(* PLC project Scenario7v1_Final.project, CODESYS CODESYS V3.5 SP5 Patch 1 *)
(* stored: creationDateTime 2014-09-12T06:04:18.7394832, modificationDateTime 2014-09-11T21:24:11.718058 *)

FUNCTION_BLOCK Magazin
  VAR_INPUT
    SliderNotMovedOut : BOOL;
    SliderMovedOut : BOOL;
    WorkpieceReady : BOOL;
    CraneDown : BOOL;
    CraneUp : BOOL;
    CraneOnConveyor : BOOL;
    CraneOnMagazin : BOOL;
    CraneSucked : BOOL;
    StartButtonMagazin : BOOL;
    SFCReset : BOOL;
    StartVar : BOOL;
  END_VAR
  VAR_OUTPUT
    CraneLower : BOOL;
    MagazinVacuumOff : BOOL;
    MagazinVacuumOn : BOOL;
    CraneTurnCounterclockwise : BOOL;
    CraneTurnClockwise : BOOL;
    MagazinSlider : BOOL;
    MagazinGreenLamp : BOOL;
    MagazinWhiteLamp : BOOL;
    StartCommandMagazin : BOOL;
  END_VAR
  VAR
    interconnectMagazinStartCommand : BOOL;
    SFCInit : BOOL;
  END_VAR

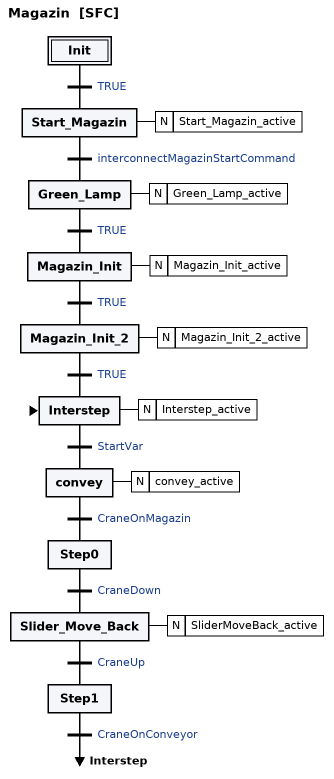
INITIAL_STEP Init:
END_STEP
TRANSITION FROM Init TO Start_Magazin
  := TRUE;
END_TRANSITION
STEP Start_Magazin:
  Start_Magazin_active(N);
END_STEP
TRANSITION FROM Start_Magazin TO Green_Lamp
  := interconnectMagazinStartCommand;
END_TRANSITION
STEP Green_Lamp:
  Green_Lamp_active(N);
END_STEP
TRANSITION FROM Green_Lamp TO Magazin_Init
  := TRUE;
END_TRANSITION
STEP Magazin_Init:
  Magazin_Init_active(N);
END_STEP
TRANSITION FROM Magazin_Init TO Magazin_Init_2
  := TRUE;
END_TRANSITION
STEP Magazin_Init_2:
  Magazin_Init_2_active(N);
END_STEP
TRANSITION FROM Magazin_Init_2 TO Interstep
  := TRUE;
END_TRANSITION
STEP Interstep:
  Interstep_active(N);
END_STEP
TRANSITION FROM Interstep TO convey
  := StartVar;
END_TRANSITION
STEP convey:
  convey_active(N);
END_STEP
TRANSITION FROM convey TO Step0
  := CraneOnMagazin;
END_TRANSITION
STEP Step0:
END_STEP
TRANSITION FROM Step0 TO Slider_Move_Back
  := CraneDown;
END_TRANSITION
STEP Slider_Move_Back:
  SliderMoveBack_active(N);
END_STEP
TRANSITION FROM Slider_Move_Back TO Step1
  := CraneUp;
END_TRANSITION
STEP Step1:
END_STEP
TRANSITION FROM Step1 TO Interstep
  := CraneOnConveyor;
END_TRANSITION

ACTION Magazin_Init_active:
                MagazinSlider := TRUE;
              
END_ACTION

ACTION Start_Magazin_active:
                MagazinSlider := FALSE;
MagazinGreenLamp := FALSE;
StartVar := FALSE;
StartCommandMagazin := FALSE;


IF(StartButtonMagazin = TRUE) THEN
	interconnectMagazinStartCommand := TRUE;
END_IF
              
END_ACTION

ACTION Green_Lamp_active:
                MagazinGreenLamp := TRUE;
interconnectMagazinStartCommand := FALSE;
              
END_ACTION

ACTION convey_active:
                IF(SliderNotMovedOut)THEN
	MagazinSlider := TRUE;
END_IF
              
END_ACTION

ACTION SliderMoveBack_active:
                IF((SliderMovedOut = TRUE)AND(SliderNotMovedOut = FALSE))THEN
	MagazinSlider := FALSE;
END_IF
              
END_ACTION

ACTION Magazin_Init_2_active:
                MagazinSlider := FALSE;
              
END_ACTION

ACTION Interstep_active:
                StartCommandMagazin := TRUE;
              
END_ACTION
END_FUNCTION_BLOCK

FUNCTION_BLOCK Stamp
  VAR_INPUT
    StampSliderSensorMovedOut : BOOL;
    StampSliderSensorMovedIn : BOOL;
    StampSliderFilled : BOOL;
    StampUp : BOOL;
    StampLowered : BOOL;
    CraneDown : BOOL;
    CraneUp : BOOL;
    CraneSucked : BOOL;
    CranePositionStamp : BOOL;
    CraneOnConveyor : BOOL;
    StampStartButton : BOOL;
    SFCReset : BOOL;
    StartVar : BOOL;
  END_VAR
  VAR_OUTPUT
    StampSliderMovedOut : BOOL;
    StampSliderMovedIn : BOOL;
    StampWhiteLamp : BOOL;
    StampPusher : BOOL;
    StampGreenLamp : BOOL;
    StampPressure : BOOL;
    StartCommandStamp : BOOL;
  END_VAR
  VAR
    interconnect : BOOL;
    Timer : TON;
    Duration : TIME := TIME#500ms;
    interconnectStampStartCommand : BOOL;
    SFCInit : BOOL;
  END_VAR

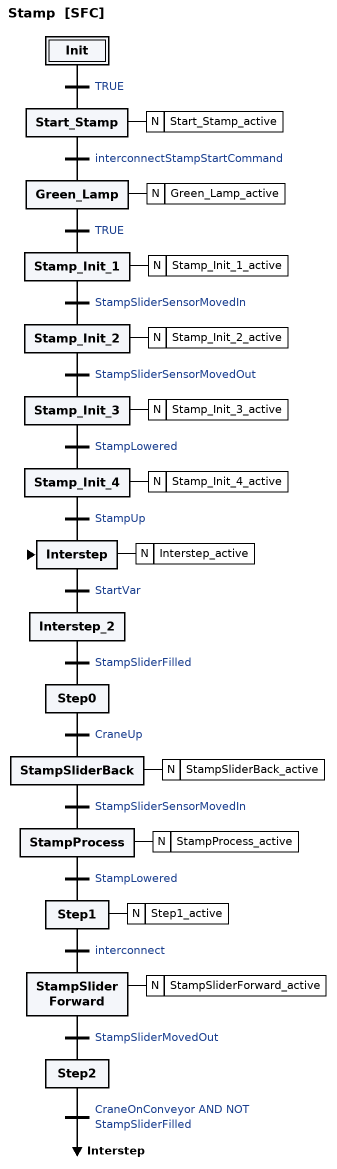
INITIAL_STEP Init:
END_STEP
TRANSITION FROM Init TO Start_Stamp
  := TRUE;
END_TRANSITION
STEP Start_Stamp:
  Start_Stamp_active(N);
END_STEP
TRANSITION FROM Start_Stamp TO Green_Lamp
  := interconnectStampStartCommand;
END_TRANSITION
STEP Green_Lamp:
  Green_Lamp_active(N);
END_STEP
TRANSITION FROM Green_Lamp TO Stamp_Init_1
  := TRUE;
END_TRANSITION
STEP Stamp_Init_1:
  Stamp_Init_1_active(N);
END_STEP
TRANSITION FROM Stamp_Init_1 TO Stamp_Init_2
  := StampSliderSensorMovedIn;
END_TRANSITION
STEP Stamp_Init_2:
  Stamp_Init_2_active(N);
END_STEP
TRANSITION FROM Stamp_Init_2 TO Stamp_Init_3
  := StampSliderSensorMovedOut;
END_TRANSITION
STEP Stamp_Init_3:
  Stamp_Init_3_active(N);
END_STEP
TRANSITION FROM Stamp_Init_3 TO Stamp_Init_4
  := StampLowered;
END_TRANSITION
STEP Stamp_Init_4:
  Stamp_Init_4_active(N);
END_STEP
TRANSITION FROM Stamp_Init_4 TO Interstep
  := StampUp;
END_TRANSITION
STEP Interstep:
  Interstep_active(N);
END_STEP
TRANSITION FROM Interstep TO Interstep_2
  := StartVar;
END_TRANSITION
STEP Interstep_2:
END_STEP
TRANSITION FROM Interstep_2 TO Step0
  := StampSliderFilled;
END_TRANSITION
STEP Step0:
END_STEP
TRANSITION FROM Step0 TO StampSliderBack
  := CraneUp;
END_TRANSITION
STEP StampSliderBack:
  StampSliderBack_active(N);
END_STEP
TRANSITION FROM StampSliderBack TO StampProcess
  := StampSliderSensorMovedIn;
END_TRANSITION
STEP StampProcess:
  StampProcess_active(N);
END_STEP
TRANSITION FROM StampProcess TO Step1
  := StampLowered;
END_TRANSITION
STEP Step1:
  Step1_active(N);
END_STEP
TRANSITION FROM Step1 TO StampSliderForward
  := interconnect;
END_TRANSITION
STEP StampSliderForward:
  StampSliderForward_active(N);
END_STEP
TRANSITION FROM StampSliderForward TO Step2
  := StampSliderMovedOut;
END_TRANSITION
STEP Step2:
END_STEP
TRANSITION FROM Step2 TO Interstep
  := CraneOnConveyor AND NOT StampSliderFilled;
END_TRANSITION

ACTION Start_Stamp_active:
                StampSliderMovedOut := FALSE;
StampSliderMovedIn := FALSE;
StampPusher := FALSE;
StampGreenLamp := FALSE;
StampPressure := FALSE;
StartCommandStamp := FALSE;


IF(StampStartButton = TRUE) THEN
	interconnectStampStartCommand := TRUE;
END_IF
              
END_ACTION

ACTION StampSliderForward_active:
                StampPusher := FALSE;
StampSliderMovedOut := TRUE;

IF((StampLowered=FALSE)AND(StampUp=TRUE))THEN
	interconnect := FALSE;
END_IF

Timer(IN:=FALSE, PT:=T#1ms);
              
END_ACTION

ACTION StampSliderBack_active:
                StampSliderMovedIn := TRUE;
StampSliderMovedOut := FALSE;
              
END_ACTION

ACTION Stamp_Init_1_active:
                StampSliderMovedIn := TRUE;
StampSliderMovedOut := FALSE;
              
END_ACTION

ACTION Step1_active:
                Timer(IN:=StampLowered, PT:=T#500MS);
interconnect := Timer.Q;
              
END_ACTION

ACTION Interstep_active:
                StartCommandStamp := TRUE;
              
END_ACTION

ACTION Green_Lamp_active:
                StampGreenLamp := TRUE;
interconnectStampStartCommand := FALSE;
              
END_ACTION

ACTION Stamp_Init_4_active:
                StampPusher := FALSE;
              
END_ACTION

ACTION Stamp_Init_3_active:
                StampPusher := TRUE;
              
END_ACTION

ACTION Stamp_Init_2_active:
                StampSliderMovedIn := FALSE;
StampSliderMovedOut := TRUE;
              
END_ACTION

ACTION StampProcess_active:
                StampSliderMovedIn := FALSE;
StampPusher := TRUE;
              
END_ACTION
END_FUNCTION_BLOCK

FUNCTION_BLOCK Crane
  VAR_INPUT
    SliderNotMovedOut : BOOL;
    SliderMovedOut : BOOL;
    MagazinCapacitiveSensor : BOOL;
    WorkpieceReady : BOOL;
    CraneDown : BOOL;
    CraneUp : BOOL;
    CraneOnConveyor : BOOL;
    CraneOnMagazin : BOOL;
    CraneSucked : BOOL;
    StampLowered : BOOL;
    CranePositionStamp : BOOL;
    MagazinOpticalSensor : BOOL;
    StampSliderFilled : BOOL;
    StartButtonMagazin : BOOL;
    SFCReset : BOOL;
    StartVar : BOOL;
    StampSliderSensorMovedOut : BOOL;
  END_VAR
  VAR_OUTPUT
    CraneLower : BOOL;
    MagazinVacuumOff : BOOL;
    MagazinVacuumOn : BOOL;
    CraneTurnCounterclockwise : BOOL;
    CraneTurnClockwise : BOOL;
    StartCommandCrane : BOOL;
  END_VAR
  VAR
    Timer1 : TON;
    Duration1 : TIME := TIME#1s500ms;
    actualtime1 : TIME;
    interconnect : BOOL;
    interconnectCraneStartCommand : BOOL;
    TimeDelay_Timer : TON;
    TimeDelay_Timer_Duration : TIME := TIME#50ms;
    TimeDelay_Timer_interconnect : BOOL;
    SFCInit : BOOL;
  END_VAR

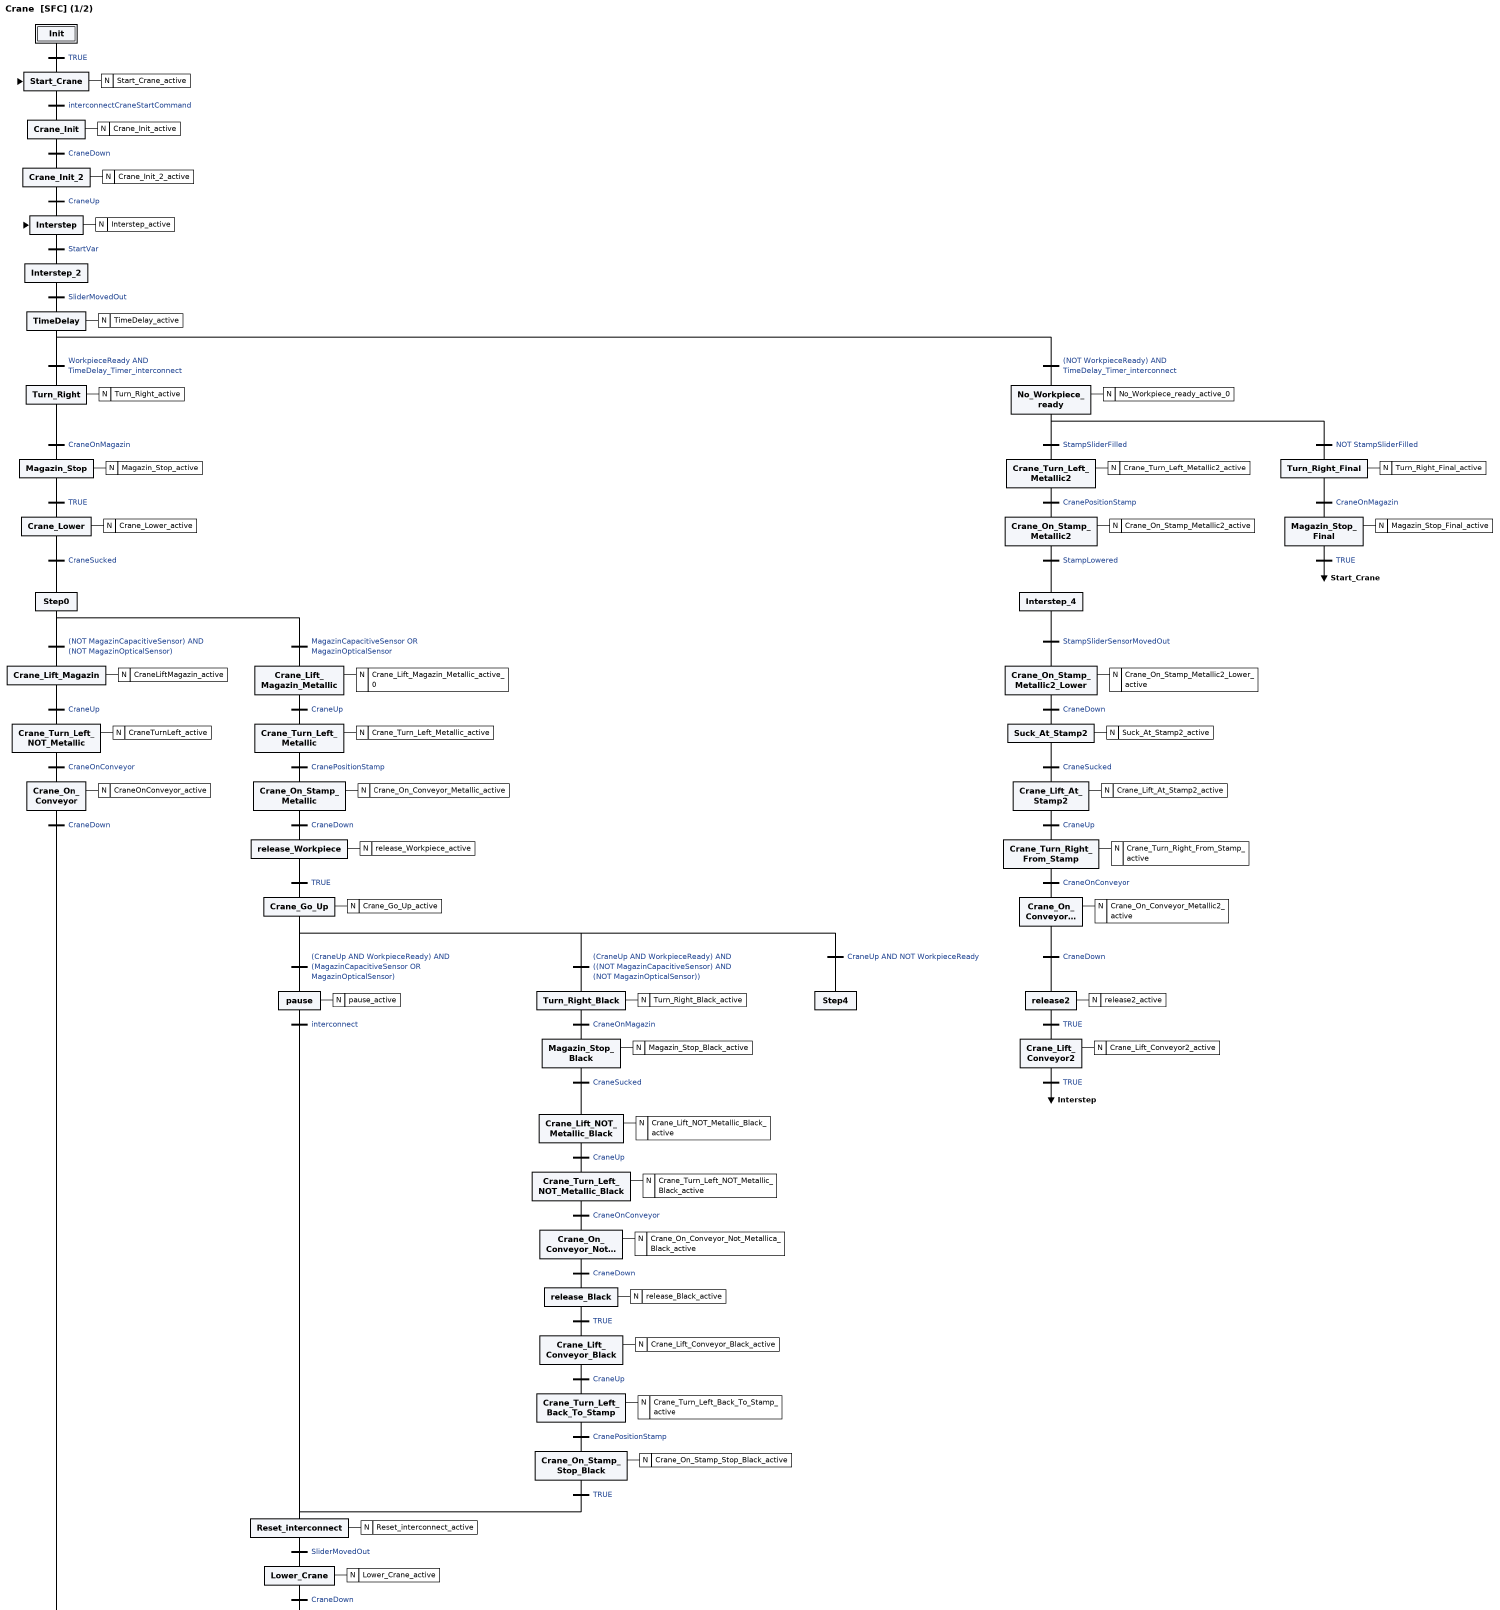
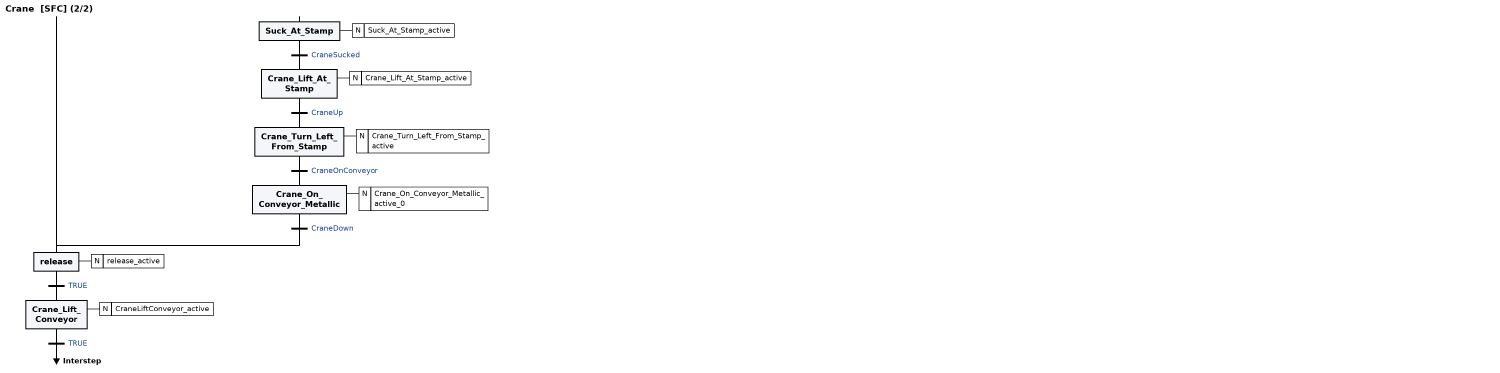
INITIAL_STEP Init:
END_STEP
TRANSITION FROM Init TO Start_Crane
  := TRUE;
END_TRANSITION
STEP Start_Crane:
  Start_Crane_active(N);
END_STEP
TRANSITION FROM Start_Crane TO Crane_Init
  := interconnectCraneStartCommand;
END_TRANSITION
STEP Crane_Init:
  Crane_Init_active(N);
END_STEP
TRANSITION FROM Crane_Init TO Crane_Init_2
  := CraneDown;
END_TRANSITION
STEP Crane_Init_2:
  Crane_Init_2_active(N);
END_STEP
TRANSITION FROM Crane_Init_2 TO Interstep
  := CraneUp;
END_TRANSITION
STEP Interstep:
  Interstep_active(N);
END_STEP
TRANSITION FROM Interstep TO Interstep_2
  := StartVar;
END_TRANSITION
STEP Interstep_2:
END_STEP
TRANSITION FROM Interstep_2 TO TimeDelay
  := SliderMovedOut;
END_TRANSITION
STEP TimeDelay:
  TimeDelay_active(N);
END_STEP
TRANSITION FROM TimeDelay TO Turn_Right
  := WorkpieceReady AND TimeDelay_Timer_interconnect;
END_TRANSITION
TRANSITION FROM TimeDelay TO No_Workpiece_ready
  := (NOT WorkpieceReady) AND TimeDelay_Timer_interconnect;
END_TRANSITION
STEP Turn_Right:
  Turn_Right_active(N);
END_STEP
TRANSITION FROM Turn_Right TO Magazin_Stop
  := CraneOnMagazin;
END_TRANSITION
STEP Magazin_Stop:
  Magazin_Stop_active(N);
END_STEP
TRANSITION FROM Magazin_Stop TO Crane_Lower
  := TRUE;
END_TRANSITION
STEP Crane_Lower:
  Crane_Lower_active(N);
END_STEP
TRANSITION FROM Crane_Lower TO Step0
  := CraneSucked;
END_TRANSITION
STEP Step0:
END_STEP
TRANSITION FROM Step0 TO Crane_Lift_Magazin
  := (NOT MagazinCapacitiveSensor) AND (NOT MagazinOpticalSensor);
END_TRANSITION
TRANSITION FROM Step0 TO Crane_Lift_Magazin_Metallic
  := MagazinCapacitiveSensor OR MagazinOpticalSensor;
END_TRANSITION
STEP Crane_Lift_Magazin:
  CraneLiftMagazin_active(N);
END_STEP
TRANSITION FROM Crane_Lift_Magazin TO Crane_Turn_Left_NOT_Metallic
  := CraneUp;
END_TRANSITION
STEP Crane_Turn_Left_NOT_Metallic:
  CraneTurnLeft_active(N);
END_STEP
TRANSITION FROM Crane_Turn_Left_NOT_Metallic TO Crane_On_Conveyor
  := CraneOnConveyor;
END_TRANSITION
STEP Crane_On_Conveyor:
  CraneOnConveyor_active(N);
END_STEP
TRANSITION FROM Crane_On_Conveyor TO release
  := CraneDown;
END_TRANSITION
STEP Crane_Lift_Magazin_Metallic:
  Crane_Lift_Magazin_Metallic_active_0(N);
END_STEP
TRANSITION FROM Crane_Lift_Magazin_Metallic TO Crane_Turn_Left_Metallic
  := CraneUp;
END_TRANSITION
STEP Crane_Turn_Left_Metallic:
  Crane_Turn_Left_Metallic_active(N);
END_STEP
TRANSITION FROM Crane_Turn_Left_Metallic TO Crane_On_Stamp_Metallic
  := CranePositionStamp;
END_TRANSITION
STEP Crane_On_Stamp_Metallic:
  Crane_On_Conveyor_Metallic_active(N);
END_STEP
TRANSITION FROM Crane_On_Stamp_Metallic TO release_Workpiece
  := CraneDown;
END_TRANSITION
STEP release_Workpiece:
  release_Workpiece_active(N);
END_STEP
TRANSITION FROM release_Workpiece TO Crane_Go_Up
  := TRUE;
END_TRANSITION
STEP Crane_Go_Up:
  Crane_Go_Up_active(N);
END_STEP
TRANSITION FROM Crane_Go_Up TO pause
  := (CraneUp AND WorkpieceReady) AND (MagazinCapacitiveSensor OR MagazinOpticalSensor);
END_TRANSITION
TRANSITION FROM Crane_Go_Up TO Turn_Right_Black
  := (CraneUp AND WorkpieceReady) AND ((NOT MagazinCapacitiveSensor) AND (NOT MagazinOpticalSensor));
END_TRANSITION
TRANSITION FROM Crane_Go_Up TO Step4
  := CraneUp AND NOT WorkpieceReady;
END_TRANSITION
STEP pause:
  pause_active(N);
END_STEP
TRANSITION FROM pause TO Reset_interconnect
  := interconnect;
END_TRANSITION
STEP Turn_Right_Black:
  Turn_Right_Black_active(N);
END_STEP
TRANSITION FROM Turn_Right_Black TO Magazin_Stop_Black
  := CraneOnMagazin;
END_TRANSITION
STEP Magazin_Stop_Black:
  Magazin_Stop_Black_active(N);
END_STEP
TRANSITION FROM Magazin_Stop_Black TO Crane_Lift_NOT_Metallic_Black
  := CraneSucked;
END_TRANSITION
STEP Crane_Lift_NOT_Metallic_Black:
  Crane_Lift_NOT_Metallic_Black_active(N);
END_STEP
TRANSITION FROM Crane_Lift_NOT_Metallic_Black TO Crane_Turn_Left_NOT_Metallic_Black
  := CraneUp;
END_TRANSITION
STEP Crane_Turn_Left_NOT_Metallic_Black:
  Crane_Turn_Left_NOT_Metallic_Black_active(N);
END_STEP
TRANSITION FROM Crane_Turn_Left_NOT_Metallic_Black TO Crane_On_Conveyor_Not_Metallica_Black
  := CraneOnConveyor;
END_TRANSITION
STEP Crane_On_Conveyor_Not_Metallica_Black:
  Crane_On_Conveyor_Not_Metallica_Black_active(N);
END_STEP
TRANSITION FROM Crane_On_Conveyor_Not_Metallica_Black TO release_Black
  := CraneDown;
END_TRANSITION
STEP release_Black:
  release_Black_active(N);
END_STEP
TRANSITION FROM release_Black TO Crane_Lift_Conveyor_Black
  := TRUE;
END_TRANSITION
STEP Crane_Lift_Conveyor_Black:
  Crane_Lift_Conveyor_Black_active(N);
END_STEP
TRANSITION FROM Crane_Lift_Conveyor_Black TO Crane_Turn_Left_Back_To_Stamp
  := CraneUp;
END_TRANSITION
STEP Crane_Turn_Left_Back_To_Stamp:
  Crane_Turn_Left_Back_To_Stamp_active(N);
END_STEP
TRANSITION FROM Crane_Turn_Left_Back_To_Stamp TO Crane_On_Stamp_Stop_Black
  := CranePositionStamp;
END_TRANSITION
STEP Crane_On_Stamp_Stop_Black:
  Crane_On_Stamp_Stop_Black_active(N);
END_STEP
TRANSITION FROM Crane_On_Stamp_Stop_Black TO Reset_interconnect
  := TRUE;
END_TRANSITION
STEP Step4:
END_STEP
STEP Reset_interconnect:
  Reset_interconnect_active(N);
END_STEP
TRANSITION FROM Reset_interconnect TO Lower_Crane
  := SliderMovedOut;
END_TRANSITION
STEP Lower_Crane:
  Lower_Crane_active(N);
END_STEP
TRANSITION FROM Lower_Crane TO Suck_At_Stamp
  := CraneDown;
END_TRANSITION
STEP Suck_At_Stamp:
  Suck_At_Stamp_active(N);
END_STEP
TRANSITION FROM Suck_At_Stamp TO Crane_Lift_At_Stamp
  := CraneSucked;
END_TRANSITION
STEP Crane_Lift_At_Stamp:
  Crane_Lift_At_Stamp_active(N);
END_STEP
TRANSITION FROM Crane_Lift_At_Stamp TO Crane_Turn_Left_From_Stamp
  := CraneUp;
END_TRANSITION
STEP Crane_Turn_Left_From_Stamp:
  Crane_Turn_Left_From_Stamp_active(N);
END_STEP
TRANSITION FROM Crane_Turn_Left_From_Stamp TO Crane_On_Conveyor_Metallic
  := CraneOnConveyor;
END_TRANSITION
STEP Crane_On_Conveyor_Metallic:
  Crane_On_Conveyor_Metallic_active_0(N);
END_STEP
TRANSITION FROM Crane_On_Conveyor_Metallic TO release
  := CraneDown;
END_TRANSITION
STEP release:
  release_active(N);
END_STEP
TRANSITION FROM release TO Crane_Lift_Conveyor
  := TRUE;
END_TRANSITION
STEP Crane_Lift_Conveyor:
  CraneLiftConveyor_active(N);
END_STEP
TRANSITION FROM Crane_Lift_Conveyor TO Interstep
  := TRUE;
END_TRANSITION
STEP No_Workpiece_ready:
  No_Workpiece_ready_active_0(N);
END_STEP
TRANSITION FROM No_Workpiece_ready TO Crane_Turn_Left_Metallic2
  := StampSliderFilled;
END_TRANSITION
TRANSITION FROM No_Workpiece_ready TO Turn_Right_Final
  := NOT StampSliderFilled;
END_TRANSITION
STEP Crane_Turn_Left_Metallic2:
  Crane_Turn_Left_Metallic2_active(N);
END_STEP
TRANSITION FROM Crane_Turn_Left_Metallic2 TO Crane_On_Stamp_Metallic2
  := CranePositionStamp;
END_TRANSITION
STEP Crane_On_Stamp_Metallic2:
  Crane_On_Stamp_Metallic2_active(N);
END_STEP
TRANSITION FROM Crane_On_Stamp_Metallic2 TO Interstep_4
  := StampLowered;
END_TRANSITION
STEP Interstep_4:
END_STEP
TRANSITION FROM Interstep_4 TO Crane_On_Stamp_Metallic2_Lower
  := StampSliderSensorMovedOut;
END_TRANSITION
STEP Crane_On_Stamp_Metallic2_Lower:
  Crane_On_Stamp_Metallic2_Lower_active(N);
END_STEP
TRANSITION FROM Crane_On_Stamp_Metallic2_Lower TO Suck_At_Stamp2
  := CraneDown;
END_TRANSITION
STEP Suck_At_Stamp2:
  Suck_At_Stamp2_active(N);
END_STEP
TRANSITION FROM Suck_At_Stamp2 TO Crane_Lift_At_Stamp2
  := CraneSucked;
END_TRANSITION
STEP Crane_Lift_At_Stamp2:
  Crane_Lift_At_Stamp2_active(N);
END_STEP
TRANSITION FROM Crane_Lift_At_Stamp2 TO Crane_Turn_Right_From_Stamp
  := CraneUp;
END_TRANSITION
STEP Crane_Turn_Right_From_Stamp:
  Crane_Turn_Right_From_Stamp_active(N);
END_STEP
TRANSITION FROM Crane_Turn_Right_From_Stamp TO Crane_On_Conveyor_Metallic2
  := CraneOnConveyor;
END_TRANSITION
STEP Crane_On_Conveyor_Metallic2:
  Crane_On_Conveyor_Metallic2_active(N);
END_STEP
TRANSITION FROM Crane_On_Conveyor_Metallic2 TO release2
  := CraneDown;
END_TRANSITION
STEP release2:
  release2_active(N);
END_STEP
TRANSITION FROM release2 TO Crane_Lift_Conveyor2
  := TRUE;
END_TRANSITION
STEP Crane_Lift_Conveyor2:
  Crane_Lift_Conveyor2_active(N);
END_STEP
TRANSITION FROM Crane_Lift_Conveyor2 TO Interstep
  := TRUE;
END_TRANSITION
STEP Turn_Right_Final:
  Turn_Right_Final_active(N);
END_STEP
TRANSITION FROM Turn_Right_Final TO Magazin_Stop_Final
  := CraneOnMagazin;
END_TRANSITION
STEP Magazin_Stop_Final:
  Magazin_Stop_Final_active(N);
END_STEP
TRANSITION FROM Magazin_Stop_Final TO Start_Crane
  := TRUE;
END_TRANSITION

ACTION Interstep_active:
                StartCommandCrane := TRUE;
              
END_ACTION

ACTION Crane_Lift_NOT_Metallic_Black_active:
                CraneLower := FALSE;
              
END_ACTION

ACTION Suck_At_Stamp_active:
                MagazinVacuumOn := TRUE;
MagazinVacuumOff := FALSE;
              
END_ACTION

ACTION Magazin_Stop_Black_active:
                CraneTurnClockwise := FALSE;
CraneTurnCounterclockwise := FALSE;
MagazinVacuumOn := TRUE;
MagazinVacuumOff := FALSE;
CraneLower := TRUE;
              
END_ACTION

ACTION Crane_On_Conveyor_Not_Metallica_Black_active:
                CraneTurnCounterclockwise := FALSE;
CraneTurnClockwise := FALSE;
CraneLower := TRUE;
              
END_ACTION

ACTION TimeDelay_active:
                TimeDelay_Timer(IN:=TRUE, PT:=TimeDelay_Timer_Duration);
TimeDelay_Timer_interconnect := TimeDelay_Timer.Q;
              
END_ACTION

ACTION Crane_Turn_Left_From_Stamp_active:
                CraneTurnClockwise := TRUE;
CraneTurnCounterclockwise := FALSE;
              
END_ACTION

ACTION CraneLiftMagazin_active:
                CraneLower := FALSE;
              
END_ACTION

ACTION Crane_Init_active:
                CraneLower := TRUE;
interconnectCraneStartCommand := FALSE;
              
END_ACTION

ACTION Magazin_Stop_Final_active:
                CraneTurnClockwise := FALSE;
CraneTurnCounterclockwise := FALSE;
              
END_ACTION

ACTION Turn_Right_Final_active:
                CraneTurnClockwise := TRUE;
CraneTurnCounterclockwise := FALSE;
              
END_ACTION

ACTION Crane_Turn_Left_Back_To_Stamp_active:
                CraneTurnCounterclockwise := TRUE;
CraneTurnClockwise := FALSE;
              
END_ACTION

ACTION Start_Crane_active:
                CraneLower := FALSE;
MagazinVacuumOff := FALSE;
MagazinVacuumOn := FALSE;
CraneTurnCounterclockwise := FALSE;
CraneTurnClockwise := FALSE;
StartVar := FALSE;
StartCommandCrane := FALSE;


IF(StartButtonMagazin = TRUE) THEN
	interconnectCraneStartCommand := TRUE;
END_IF
              
END_ACTION

ACTION Crane_On_Stamp_Metallic2_active:
                CraneTurnCounterclockwise := FALSE;
CraneTurnClockwise := FALSE;
              
END_ACTION

ACTION Crane_On_Stamp_Metallic2_Lower_active:
                CraneLower := TRUE;
              
END_ACTION

ACTION Crane_Turn_Left_Metallic_active:
                CraneTurnCounterclockwise := TRUE;
CraneTurnClockwise := FALSE;
              
END_ACTION

ACTION release2_active:
                MagazinVacuumOff := TRUE;
MagazinVacuumOn := FALSE;
              
END_ACTION

ACTION CraneOnConveyor_active:
                CraneTurnCounterclockwise := FALSE;
CraneTurnClockwise := FALSE;
CraneLower := TRUE;
              
END_ACTION

ACTION Crane_On_Conveyor_Metallic2_active:
                CraneTurnCounterclockwise := FALSE;
CraneTurnClockwise := FALSE;
CraneLower := TRUE;
              
END_ACTION

ACTION Crane_Turn_Right_From_Stamp_active:
                CraneTurnClockwise := TRUE;
CraneTurnCounterclockwise := FALSE;
              
END_ACTION

ACTION Reset_interconnect_active:
                interconnect := FALSE;
Timer1(IN:=FALSE,PT:=T#1ms);
              
END_ACTION

ACTION Crane_Turn_Left_Metallic2_active:
                CraneTurnCounterclockwise := TRUE;
CraneTurnClockwise := FALSE;
              
END_ACTION

ACTION Turn_Right_active:
                CraneTurnClockwise := TRUE;
CraneTurnCounterclockwise := FALSE;
              
END_ACTION

ACTION Crane_Lift_Magazin_Metallic_active_0:
                CraneLower := FALSE;
              
END_ACTION

ACTION release_Black_active:
                MagazinVacuumOn := FALSE;
MagazinVacuumOff := TRUE;
              
END_ACTION

ACTION Lower_Crane_active:
                CraneLower := TRUE;
              
END_ACTION

ACTION release_Workpiece_active:
                MagazinVacuumOff := TRUE;
MagazinVacuumOn := FALSE;
              
END_ACTION

ACTION No_Workpiece_ready_active_0:
                MagazinVacuumOn := FALSE;
MagazinVacuumOff := FALSE;
CraneLower := FALSE;

              
END_ACTION

ACTION Crane_Lift_At_Stamp_active:
                CraneLower := FALSE;
              
END_ACTION

ACTION Crane_Go_Up_active:
                CraneLower := FALSE;
              
END_ACTION

ACTION pause_active:
                Timer1(IN:=CraneUp, PT:=Duration1);
interconnect := Timer1.Q;
              
END_ACTION

ACTION Crane_Lift_Conveyor2_active:
                CraneLower := FALSE;
              
END_ACTION

ACTION Crane_Turn_Left_NOT_Metallic_Black_active:
                CraneTurnCounterclockwise := TRUE;
CraneTurnClockwise := FALSE;
              
END_ACTION

ACTION Crane_On_Conveyor_Metallic_active:
                CraneTurnCounterclockwise := FALSE;
CraneTurnClockwise := FALSE;
CraneLower := TRUE;
              
END_ACTION

ACTION Magazin_Stop_active:
                CraneTurnClockwise := FALSE;
CraneTurnCounterclockwise := FALSE;
              
END_ACTION

ACTION Suck_At_Stamp2_active:
                MagazinVacuumOn := TRUE;
MagazinVacuumOff := FALSE;
              
END_ACTION

ACTION CraneLiftConveyor_active:
                CraneLower := FALSE;
              
END_ACTION

ACTION Turn_Right_Black_active:
                CraneTurnClockwise := TRUE;
CraneTurnCounterclockwise := FALSE;
              
END_ACTION

ACTION Crane_On_Stamp_Stop_Black_active:
                CraneTurnClockwise := FALSE;
CraneTurnCounterclockwise := FALSE;
              
END_ACTION

ACTION CraneTurnLeft_active:
                CraneTurnCounterclockwise := TRUE;
CraneTurnClockwise := FALSE;
              
END_ACTION

ACTION release_active:
                MagazinVacuumOff := TRUE;
MagazinVacuumOn := FALSE;
              
END_ACTION

ACTION Crane_Lower_active:
                MagazinVacuumOn := TRUE;
MagazinVacuumOff := FALSE;
CraneLower := TRUE;
              
END_ACTION

ACTION Crane_Lift_Conveyor_Black_active:
                CraneLower := FALSE;
              
END_ACTION

ACTION Crane_Lift_At_Stamp2_active:
                CraneLower := FALSE;
              
END_ACTION

ACTION Crane_On_Conveyor_Metallic_active_0:
                CraneTurnCounterclockwise := FALSE;
CraneTurnClockwise := FALSE;
CraneLower := TRUE;
              
END_ACTION

ACTION Crane_Init_2_active:
                CraneLower := FALSE;
              
END_ACTION
END_FUNCTION_BLOCK

PROGRAM Main
  VAR
    Sensor_StartButtonMagazin : BOOL;
    Sensor_MagazinEmergencyStop : BOOL;
    Sensor_MagazinSwitchManuellAutomatic : BOOL;
    Sensor_CraneSucked : BOOL;
    Sensor_CraneDown : BOOL;
    Sensor_CraneUp : BOOL;
    Sensor_SliderNotMovedOut : BOOL;
    Sensor_SliderMovedOut : BOOL;
    Sensor_MagazinCapacitiveSensor : BOOL;
    Sensor_MagazinOpticalSensor : BOOL;
    Sensor_CranePositionStamp : BOOL;
    Sensor_CraneOnConveyor : BOOL;
    Sensor_CraneOnMagazin : BOOL;
    Sensor_WorkpieceReady : BOOL;
    Sensor_CranePosition : BOOL;
    Sensor_StampSliderSensorMovedOut : BOOL;
    Sensor_StampSliderSensorMovedIn : BOOL;
    Sensor_StampSliderFilled : BOOL;
    Sensor_StampUp : BOOL;
    Sensor_StampLowered : BOOL;
    Sensor_StampSwitchManuellAutomatic : BOOL;
    Sensor_StampEmergencyStop : BOOL;
    Sensor_StampStartButton : BOOL;
    Actuator_MagazinSlider : BOOL;
    Actuator_CraneLower : BOOL;
    Actuator_MagazinVacuumOn : BOOL;
    Actuator_MagazinVacuumOff : BOOL;
    Actuator_MagazinGreenLamp : BOOL;
    Actuator_MagazinWhiteLamp : BOOL;
    Actuator_CraneTurnCounterclockwise : BOOL;
    Actuator_CraneTurnClockwise : BOOL;
    Actuator_StampSliderMovedOut : BOOL;
    Actuator_StampSliderMovedIn : BOOL;
    Actuator_StampWhiteLamp : BOOL;
    Actuator_StampGreenLamp : BOOL;
    Actuator_StampPusher : BOOL;
    Actuator_AnalogCranePressure : INT;
    Mag : Magazin;
    Crane : Crane;
    Stamp : Stamp;
  END_VAR

            Mag.SliderNotMovedOut := Sensor_SliderNotMovedOut;
Mag.SliderMovedOut := Sensor_SliderMovedOut;
Mag.CraneOnMagazin := Sensor_CraneOnMagazin;
Mag.CraneDown := Sensor_CraneDown;
Mag.CraneUp := Sensor_CraneUp;
Mag.CraneOnConveyor := Sensor_CraneOnConveyor;
Mag.WorkpieceReady := Sensor_WorkpieceReady;
Mag.StartButtonMagazin := Sensor_StartButtonMagazin;

Actuator_MagazinSlider := Mag.MagazinSlider;
Actuator_MagazinGreenLamp := Mag.MagazinGreenLamp;

Crane.CraneUp := Sensor_CraneUp;
Crane.CraneOnConveyor := Sensor_CraneOnConveyor;
Crane.CraneDown := Sensor_CraneDown;
Crane.CraneSucked := Sensor_CraneSucked;
Crane.CraneOnMagazin := Sensor_CraneOnMagazin;
Crane.MagazinCapacitiveSensor := Sensor_MagazinCapacitiveSensor;
Crane.CranePositionStamp := Sensor_CranePositionStamp;
Crane.SliderMovedOut := Sensor_SliderMovedOut;
Crane.WorkpieceReady := Sensor_WorkpieceReady;
Crane.MagazinOpticalSensor := Sensor_MagazinOpticalSensor;
Crane.StampSliderFilled := Sensor_StampSliderFilled;
Crane.StampSliderSensorMovedOut := Sensor_StampSliderSensorMovedOut;
Crane.StampLowered := Sensor_StampLowered;
Crane.StartButtonMagazin := Sensor_StartButtonMagazin;

Actuator_CraneTurnCounterclockwise := Crane.CraneTurnCounterclockwise;
Actuator_CraneTurnClockwise := Crane.CraneTurnClockwise;
Actuator_CraneLower := Crane.CraneLower;
Actuator_MagazinVacuumOff := Crane.MagazinVacuumOff;
Actuator_MagazinVacuumOn := Crane.MagazinVacuumOn;

Stamp.StampSliderSensorMovedOut := Sensor_StampSliderSensorMovedOut;
Stamp.StampSliderSensorMovedIn := Sensor_StampSliderSensorMovedIn;
Stamp.StampSliderFilled := Sensor_StampSliderFilled;
Stamp.StampUp := Sensor_StampUp;
Stamp.StampLowered := Sensor_StampLowered;
Stamp.CraneDown := Sensor_CraneDown;
Stamp.CraneUp := Sensor_CraneUp;
Stamp.CraneSucked := Sensor_CraneSucked;
Stamp.CranePositionStamp := Sensor_CranePositionStamp;
Stamp.CraneOnConveyor := Sensor_CraneOnConveyor;
Stamp.StampStartButton := Sensor_StampStartButton;

Actuator_StampSliderMovedOut := Stamp.StampSliderMovedOut;
Actuator_StampSliderMovedIn := Stamp.StampSliderMovedIn;
Actuator_StampWhiteLamp := Stamp.StampWhiteLamp;
Actuator_StampPusher := Stamp.StampPusher;
Actuator_StampGreenLamp := Stamp.StampGreenLamp;

Actuator_AnalogCranePressure := 6000;


IF((Sensor_StampEmergencyStop) AND (Sensor_MagazinEmergencyStop))THEN
	Mag();
	Crane();
	Stamp();
	IF((Actuator_MagazinGreenLamp) AND (Actuator_StampGreenLamp))THEN
		IF((Stamp.StartCommandStamp) AND (Crane.StartCommandCrane) AND (Mag.StartCommandMagazin))THEN
			Crane.StartVar := TRUE;
			Mag.StartVar := TRUE;
			Stamp.StartVar := TRUE;
		END_IF
	END_IF
	Crane.SFCReset := FALSE;
	Mag.SFCReset := FALSE;
	Stamp.SFCReset := FALSE;
ELSIF ((NOT Sensor_StampEmergencyStop) OR (NOT Sensor_MagazinEmergencyStop))THEN
	Actuator_MagazinSlider := FALSE;
	Actuator_CraneLower := FALSE;
	Actuator_MagazinVacuumOn := FALSE;
	Actuator_MagazinVacuumOff := TRUE;
	Actuator_MagazinGreenLamp := FALSE;
	Actuator_CraneTurnCounterclockwise := FALSE;
	Actuator_CraneTurnClockwise := FALSE;
	Actuator_StampSliderMovedOut := TRUE;
	Actuator_StampSliderMovedIn := FALSE;
	Actuator_StampGreenLamp := FALSE;
	Actuator_StampPusher := FALSE;

	Actuator_AnalogCranePressure := 0;
	
	Crane.SFCReset := TRUE;
	Mag.SFCReset := TRUE;
	Stamp.SFCReset := TRUE;
	
	Crane.StartVar := FALSE;
	Mag.StartVar := FALSE;
	Stamp.StartVar := FALSE;
END_IF
          
END_PROGRAM
